// TIA Portal project "Sistema_Irrigazione2" (V15.1)

(* hardware
DEVICE "S7-1200 station_1"  S7-1200 Station
   slot 0: "Telaio di montaggio_0"  S7-1200 Rack  Rack  V1.0
   slot 1: "PLC_1"  CPU 1214C DC/DC/DC  6ES7 214-1AG40-0XB0  V4.2
*)

// ===== PLC "PLC_1"  CPU 1214C DC/DC/DC =====

VAR_GLOBAL   // PLC tag table "Tabella delle variabili standard"
   "sec" AT %I0.0 : Bool;
   "fine_timer" AT %M0.0 : Bool;
   "fine_primo" AT %M0.1 : Bool;
   "fine_secondo" AT %M0.2 : Bool;
   "fine_terzo" AT %M0.3 : Bool;
   "fine_quarto" AT %M0.4 : Bool;
   "apri1" AT %Q0.0 : Bool;
   "chiudi1" AT %Q0.1 : Bool;
   "apri2" AT %Q0.2 : Bool;
   "chiudi2" AT %Q0.3 : Bool;
   "apri3" AT %Q0.4 : Bool;
   "chiudi3" AT %Q0.5 : Bool;
   "apri4" AT %Q0.6 : Bool;
   "chiudi4" AT %Q0.7 : Bool;
END_VAR

VAR_GLOBAL CONSTANT   // PLC tag table "Tabella delle variabili standard"
   "intervalloIrrigazione" : Time := T#60s;
   "DurataApertura" : Time := T#4s;
   "DurataChiusura" : Time := T#2s;
   "DurataIrrigazioneRamo" : Time := T#10s;
END_VAR

DATA_BLOCK "variabili_stato"   // DB1
{ S7_Optimized_Access := 'TRUE' }
VERSION : 0.1
   VAR RETAIN
      home : Bool := true;
      primo : Bool;
      secondo : Bool;
      terzo : Bool;
      quarto : Bool;
   END_VAR
BEGIN
END_DATA_BLOCK

DATA_BLOCK "ramo_irrigazione_DB"   // DB4
{ S7_Optimized_Access := 'TRUE' }
VERSION : 0.1
// stored: InstanceOfName ramo_irrigazione
"ramo_irrigazione"
BEGIN
END_DATA_BLOCK

DATA_BLOCK "ramo_irrigazione_DB_1"   // DB5
{ S7_Optimized_Access := 'TRUE' }
VERSION : 0.1
// stored: InstanceOfName ramo_irrigazione
"ramo_irrigazione"
BEGIN
END_DATA_BLOCK

DATA_BLOCK "ramo_irrigazione_DB_2"   // DB6
{ S7_Optimized_Access := 'TRUE' }
VERSION : 0.1
// stored: InstanceOfName ramo_irrigazione
"ramo_irrigazione"
BEGIN
END_DATA_BLOCK

DATA_BLOCK "ramo_irrigazione_DB_3"   // DB7
{ S7_Optimized_Access := 'TRUE' }
VERSION : 0.1
// stored: InstanceOfName ramo_irrigazione
"ramo_irrigazione"
BEGIN
END_DATA_BLOCK

// folder: System blocks/Program resources

DATA_BLOCK "IEC_Timer_0_DB"   // DB2
{ S7_Optimized_Access := 'TRUE' }
AUTHOR : Simatic
FAMILY : IEC
NAME : IEC_TMR
VERSION : 1.0
// stored: InstanceOfName IEC_TIMER
"IEC_TIMER"
BEGIN
END_DATA_BLOCK

DATA_BLOCK "IEC_Timer_0_DB_1"   // DB3
{ S7_Optimized_Access := 'TRUE' }
AUTHOR : Simatic
FAMILY : IEC
NAME : IEC_TMR
VERSION : 1.0
// stored: InstanceOfName IEC_TIMER
"IEC_TIMER"
BEGIN
END_DATA_BLOCK

// folder: (top level)

FUNCTION_BLOCK "ramo_irrigazione"   // FB1, LAD
{ S7_Optimized_Access := 'TRUE' }
VERSION : 0.1
   VAR_INPUT
      tempoApertura : Time := T#20s;
      tempoChiusura : Time := T#20s;
      tempoIrrigazione : Time := T#20s;
      Abilitazione : Bool;
   END_VAR
   VAR_OUTPUT
      comandoApertura : Bool;
      comandoChiusura : Bool;
      Completato : Bool;
   END_VAR
   VAR RETAIN
      home : Bool := true;
      apri : Bool;
      irriga : Bool;
      chiudi : Bool;
      fine : Bool;
   END_VAR
   VAR_TEMP
      temp : Bool;
   END_VAR
   VAR_TEMP   // added for the SCL form of the ladder/FBD networks
      _w1 : Bool;
   END_VAR
BEGIN

REGION Network 1
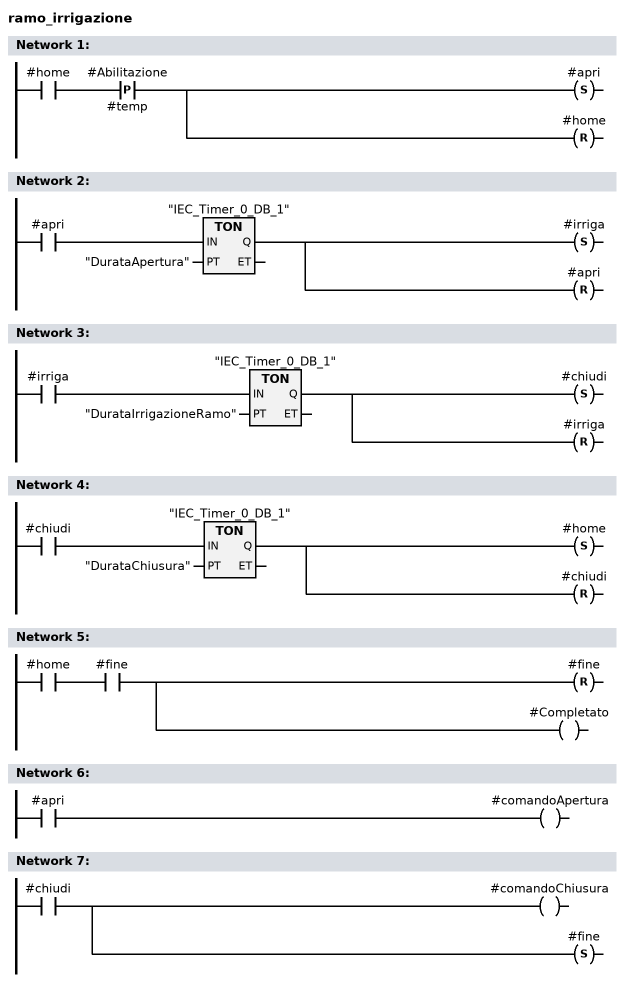
   RUNG wire#powerrail
      Contact( #home )
      P_Contact(operand := #Abilitazione, bit := #temp)
      wire#w1
      S_Coil( #apri )
   END_RUNG
   RUNG wire#w1
      R_Coil( #home )
   END_RUNG
   // the same network as SCL:
   #_w1 := #home AND #Abilitazione AND NOT #temp;   // rising edge of #Abilitazione
   #temp := #Abilitazione;
   IF #_w1 THEN
       #apri := TRUE;
       #home := FALSE;
   END_IF;
END_REGION

REGION Network 2
   "IEC_Timer_0_DB_1".TON(IN := #apri, PT := "DurataApertura");
   IF "IEC_Timer_0_DB_1".Q THEN
       #irriga := TRUE;
       #apri := FALSE;
   END_IF;
END_REGION

REGION Network 3
   "IEC_Timer_0_DB_1".TON(IN := #irriga, PT := "DurataIrrigazioneRamo");
   IF "IEC_Timer_0_DB_1".Q THEN
       #chiudi := TRUE;
       #irriga := FALSE;
   END_IF;
END_REGION

REGION Network 4
   "IEC_Timer_0_DB_1".TON(IN := #chiudi, PT := "DurataChiusura");
   IF "IEC_Timer_0_DB_1".Q THEN
       #home := TRUE;
       #chiudi := FALSE;
   END_IF;
END_REGION

REGION Network 5
   RUNG wire#powerrail
      Contact( #home )
      Contact( #fine )
      wire#w1
      R_Coil( #fine )
   END_RUNG
   RUNG wire#w1
      Coil( #Completato )
   END_RUNG
   // the same network as SCL:
   #_w1 := #home AND #fine;
   IF #_w1 THEN #fine := FALSE; END_IF;
   #Completato := #_w1;
END_REGION

REGION Network 6
   RUNG wire#powerrail
      Contact( #apri )
      Coil( #comandoApertura )
   END_RUNG
   // the same network as SCL:
   #comandoApertura := #apri;
END_REGION

REGION Network 7
   RUNG wire#powerrail
      Contact( #chiudi )
      wire#w1
      Coil( #comandoChiusura )
   END_RUNG
   RUNG wire#w1
      S_Coil( #fine )
   END_RUNG
   // the same network as SCL:
   #comandoChiusura := #chiudi;
   IF #chiudi THEN #fine := TRUE; END_IF;
END_REGION
END_FUNCTION_BLOCK

ORGANIZATION_BLOCK "Main"   // OB1, LAD, ProgramCycle
TITLE = "Main Program Sweep (Cycle)"
{ S7_Optimized_Access := 'TRUE' }
VERSION : 0.1
   VAR_INPUT
      Initial_Call : Bool;   // Initial call of this OB
      Remanence : Bool;   // =True, if remanent data are available
   END_VAR
BEGIN

REGION Network 1
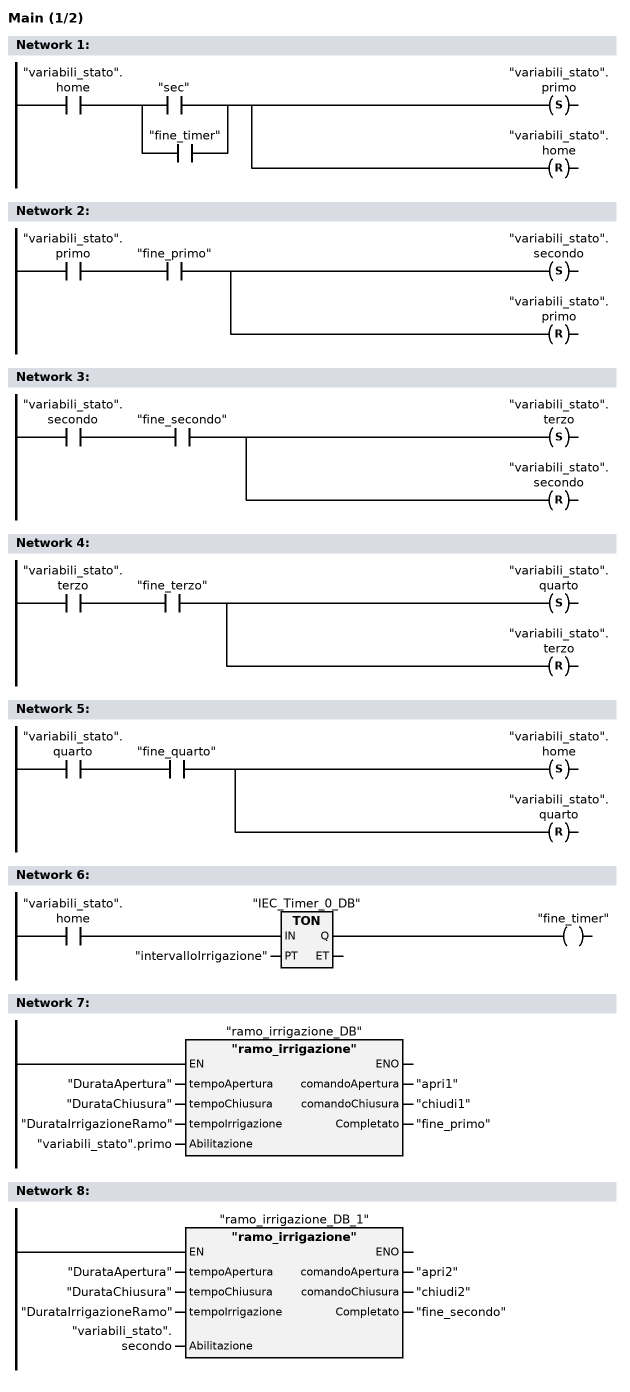
   RUNG wire#powerrail
      Contact( "variabili_stato".home )
      wire#w1
      Contact( "sec" )
      wire#w2
      S_Coil( "variabili_stato".primo )
   END_RUNG
   RUNG wire#w1
      Contact( "fine_timer" )
   END_RUNG wire#w2
   RUNG wire#w2
      R_Coil( "variabili_stato".home )
   END_RUNG
   // the same network as SCL:
   IF "variabili_stato".home AND ("sec" OR "fine_timer") THEN
       "variabili_stato".primo := TRUE;
       "variabili_stato".home := FALSE;
   END_IF;
END_REGION

REGION Network 2
   RUNG wire#powerrail
      Contact( "variabili_stato".primo )
      Contact( "fine_primo" )
      wire#w1
      S_Coil( "variabili_stato".secondo )
   END_RUNG
   RUNG wire#w1
      R_Coil( "variabili_stato".primo )
   END_RUNG
   // the same network as SCL:
   IF "variabili_stato".primo AND "fine_primo" THEN
       "variabili_stato".secondo := TRUE;
       "variabili_stato".primo := FALSE;
   END_IF;
END_REGION

REGION Network 3
   RUNG wire#powerrail
      Contact( "variabili_stato".secondo )
      Contact( "fine_secondo" )
      wire#w1
      S_Coil( "variabili_stato".terzo )
   END_RUNG
   RUNG wire#w1
      R_Coil( "variabili_stato".secondo )
   END_RUNG
   // the same network as SCL:
   IF "variabili_stato".secondo AND "fine_secondo" THEN
       "variabili_stato".terzo := TRUE;
       "variabili_stato".secondo := FALSE;
   END_IF;
END_REGION

REGION Network 4
   RUNG wire#powerrail
      Contact( "variabili_stato".terzo )
      Contact( "fine_terzo" )
      wire#w1
      S_Coil( "variabili_stato".quarto )
   END_RUNG
   RUNG wire#w1
      R_Coil( "variabili_stato".terzo )
   END_RUNG
   // the same network as SCL:
   IF "variabili_stato".terzo AND "fine_terzo" THEN
       "variabili_stato".quarto := TRUE;
       "variabili_stato".terzo := FALSE;
   END_IF;
END_REGION

REGION Network 5
   RUNG wire#powerrail
      Contact( "variabili_stato".quarto )
      Contact( "fine_quarto" )
      wire#w1
      S_Coil( "variabili_stato".home )
   END_RUNG
   RUNG wire#w1
      R_Coil( "variabili_stato".quarto )
   END_RUNG
   // the same network as SCL:
   IF "variabili_stato".quarto AND "fine_quarto" THEN
       "variabili_stato".home := TRUE;
       "variabili_stato".quarto := FALSE;
   END_IF;
END_REGION

REGION Network 6
   "IEC_Timer_0_DB".TON(IN := "variabili_stato".home, PT := "intervalloIrrigazione");
   "fine_timer" := "IEC_Timer_0_DB".Q;
END_REGION

REGION Network 7
   RUNG wire#powerrail
      "ramo_irrigazione_DB"(tempoApertura := "DurataApertura", tempoChiusura := "DurataChiusura", tempoIrrigazione := "DurataIrrigazioneRamo", Abilitazione := "variabili_stato".primo, comandoApertura => "apri1", comandoChiusura => "chiudi1", Completato => "fine_primo")
   END_RUNG
   // the same network as SCL:
   "ramo_irrigazione_DB"(tempoApertura := "DurataApertura",   // "ramo_irrigazione"
                         tempoChiusura := "DurataChiusura",
                         tempoIrrigazione := "DurataIrrigazioneRamo",
                         Abilitazione := "variabili_stato".primo,
                         comandoApertura => "apri1",
                         comandoChiusura => "chiudi1",
                         Completato => "fine_primo");
END_REGION

REGION Network 8
   RUNG wire#powerrail
      "ramo_irrigazione_DB_1"(tempoApertura := "DurataApertura", tempoChiusura := "DurataChiusura", tempoIrrigazione := "DurataIrrigazioneRamo", Abilitazione := "variabili_stato".secondo, comandoApertura => "apri2", comandoChiusura => "chiudi2", Completato => "fine_secondo")
   END_RUNG
   // the same network as SCL:
   "ramo_irrigazione_DB_1"(tempoApertura := "DurataApertura",   // "ramo_irrigazione"
                           tempoChiusura := "DurataChiusura",
                           tempoIrrigazione := "DurataIrrigazioneRamo",
                           Abilitazione := "variabili_stato".secondo,
                           comandoApertura => "apri2",
                           comandoChiusura => "chiudi2",
                           Completato => "fine_secondo");
END_REGION

REGION Network 9
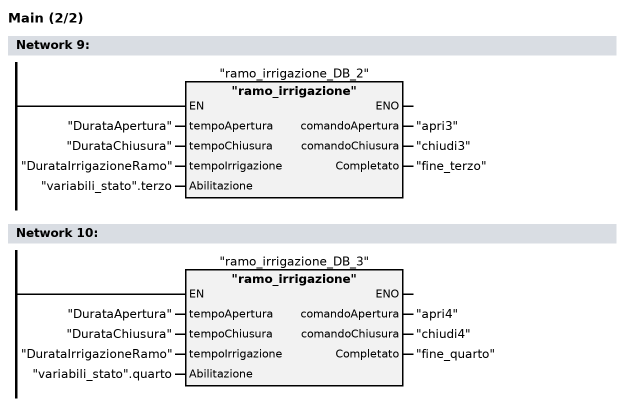
   RUNG wire#powerrail
      "ramo_irrigazione_DB_2"(tempoApertura := "DurataApertura", tempoChiusura := "DurataChiusura", tempoIrrigazione := "DurataIrrigazioneRamo", Abilitazione := "variabili_stato".terzo, comandoApertura => "apri3", comandoChiusura => "chiudi3", Completato => "fine_terzo")
   END_RUNG
   // the same network as SCL:
   "ramo_irrigazione_DB_2"(tempoApertura := "DurataApertura",   // "ramo_irrigazione"
                           tempoChiusura := "DurataChiusura",
                           tempoIrrigazione := "DurataIrrigazioneRamo",
                           Abilitazione := "variabili_stato".terzo,
                           comandoApertura => "apri3",
                           comandoChiusura => "chiudi3",
                           Completato => "fine_terzo");
END_REGION

REGION Network 10
   RUNG wire#powerrail
      "ramo_irrigazione_DB_3"(tempoApertura := "DurataApertura", tempoChiusura := "DurataChiusura", tempoIrrigazione := "DurataIrrigazioneRamo", Abilitazione := "variabili_stato".quarto, comandoApertura => "apri4", comandoChiusura => "chiudi4", Completato => "fine_quarto")
   END_RUNG
   // the same network as SCL:
   "ramo_irrigazione_DB_3"(tempoApertura := "DurataApertura",   // "ramo_irrigazione"
                           tempoChiusura := "DurataChiusura",
                           tempoIrrigazione := "DurataIrrigazioneRamo",
                           Abilitazione := "variabili_stato".quarto,
                           comandoApertura => "apri4",
                           comandoChiusura => "chiudi4",
                           Completato => "fine_quarto");
END_REGION
END_ORGANIZATION_BLOCK